FUNCTION_BLOCK FB_FieldCodecFixed32 IMPLEMENTS I_FieldCodec
VAR_INPUT
END_VAR
VAR_OUTPUT
END_VAR
VAR
    nValue : UDINT;
END_VAR

METHOD IsPackedRepeatedField : BOOL
VAR_INPUT
	nTag	: UDINT;
END_VAR
IsPackedRepeatedField := F_IsPackedRepeatedField(nTag);
END_METHOD


METHOD ValueReader : HRESULT
VAR_IN_OUT CONSTANT
	aBuffer	: ARRAY [*] OF BYTE;
END_VAR
VAR_IN_OUT
	stState	: ST_ParserInternalState;
END_VAR
VAR_OUTPUT
	anyOut	: T_Any;
END_VAR

ValueReader := F_ParseRawLittleEndian32(aBuffer, stState, nValue=> nValue);
anyOut := F_ToAnyType(anyArg:= nValue);
END_METHOD

{warning 'Add method implementation '}
{attribute 'analysis' := '-33'}
METHOD ValueWriter : HRESULT
VAR_IN_OUT
	aBuffer	: ARRAY [*] OF BYTE;
END_VAR
VAR_IN_OUT
	stState	: ST_WriterInternalState;
END_VAR
VAR_INPUT
	anyIn	: ANY;
END_VAR
END_METHOD

END_FUNCTION_BLOCK

(* stored: Version 1.1.0.1
   POU FB_FieldCodecFixed32: Id {38901a8e-394b-4d55-8a74-7207a14e063d}, SpecialFunc None
   Method IsPackedRepeatedField: Id {a1f6734c-c045-4396-8001-d851a3e88625}
   Method ValueReader: Id {c1844dc8-2aa4-44a1-8a79-d239b818953a}
   Method ValueWriter: Id {048a0cbc-dc70-44aa-9dc1-035dba44512b} *)
